// TIA Portal project "Project1" (V16)

(* hardware
DEVICE "S7300/ET200M station_1"  S7-300 station
   slot 0: "Rail_0"  Rail  6ES7 390-1***0-0AA0
   slot 2: "PLC_1"  CPU 315-2 PN/DP  6ES7 315-2EH14-0AB0  V3.2
      slot 2: "PROFINET interface_1"  PN-IO
         slot 1: "Port_1"  Port
         slot 2: "Port_2"  Port
*)

// ===== PLC "PLC_1"  CPU 315-2 PN/DP =====

VAR_GLOBAL   // PLC tag table "Default tag table"
   "Tag_1" AT %I0.0 : Bool;
   "Tag_2" AT %I0.1 : Bool;
   "Tag_3" AT %Q0.0 : Bool;
   "Tag_4" AT %I0.2 : Bool;
   "Tag_5" AT %I0.3 : Bool;
   "Tag_6" AT %M0.0 : Bool;
   "Tag_7" AT %Q0.2 : Bool;
END_VAR

ORGANIZATION_BLOCK "Main"   // OB1, LAD
TITLE = "Main Program Sweep (Cycle)"
{ S7_Optimized_Access := 'FALSE' }
VERSION : 0.1
   VAR_TEMP
      OB1_EV_CLASS : Byte;   // Bits 0-3 = 1 (Coming event), Bits 4-7 = 1 (Event class 1)
      OB1_SCAN_1 : Byte;   // 1 (Cold restart scan 1 of OB 1), 3 (Scan 2-n of OB 1)
      OB1_PRIORITY : Byte;   // Priority of OB Execution
      OB1_OB_NUMBR : Byte;   // 1 (Organization block 1, OB1)
      OB1_RESERVED_1 : Byte;   // Reserved for system
      OB1_RESERVED_2 : Byte;   // Reserved for system
      OB1_PREV_CYCLE : Int;   // Cycle time of previous OB1 scan (milliseconds)
      OB1_MIN_CYCLE : Int;   // Minimum cycle time of OB1 (milliseconds)
      OB1_MAX_CYCLE : Int;   // Maximum cycle time of OB1 (milliseconds)
      OB1_DATE_TIME : Date_And_Time;   // Date and time OB1 started
   END_VAR
BEGIN

REGION Network 1: Exclusive OR
   // Exclusive OR
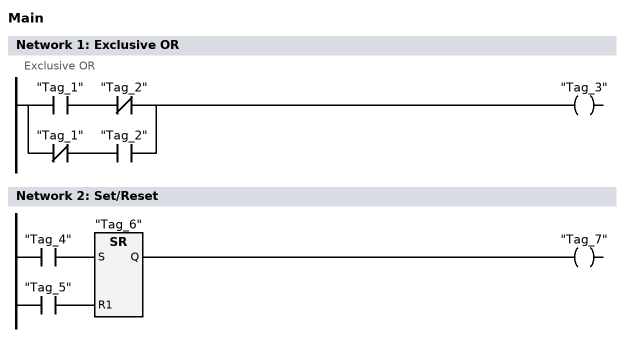
   RUNG wire#powerrail
      Contact( "Tag_1" )
      I_Contact( "Tag_2" )
      wire#w1
      Coil( "Tag_3" )
   END_RUNG
   RUNG wire#powerrail
      I_Contact( "Tag_1" )
      Contact( "Tag_2" )
   END_RUNG wire#w1
   // the same network as SCL:
   "Tag_3" := ("Tag_1" AND NOT "Tag_2") OR (NOT "Tag_1" AND "Tag_2");
END_REGION

REGION Network 2: Set/Reset
   RUNG wire#powerrail
      Contact( "Tag_4" )
      S_SR(operand := "Tag_6", r1 := wire#w1)
      Coil( "Tag_7" )
   END_RUNG
   RUNG wire#powerrail
      Contact( "Tag_5" )
   END_RUNG wire#w1
   // the same network as SCL:
   IF "Tag_4" THEN
       "Tag_6" := TRUE;   // SR flip-flop
   END_IF;
   IF "Tag_5" THEN "Tag_6" := FALSE; END_IF;
   "Tag_7" := "Tag_6";
END_REGION
END_ORGANIZATION_BLOCK